TYPE ST_Variable :
STRUCT
	Value				:REAL;
	Description			:STRING(100);
END_STRUCT
END_TYPE

(* stored: Version 1.1.0.1, ProductVersion 3.1.4024.3
   DUT ST_Variable: Id {d534504e-2387-4c6c-abc8-8011d3ef165a} *)
